VISUALIZATION Visualization_1  // 2x2
END_VISUALIZATION

(* stored: Version 1.1.0.1, ProductVersion 3.1.4024.2
   Visu Visualization_1: Id {c01c1f05-1876-4b1c-80af-af6a80a21984} *)
